		40120: 	
			SCREWING_RESULT:=E_TEST_STATE.PASSED;
			IF SCREWING_RESULT=E_TEST_STATE.PASSED THEN
				STATE:=40130;
			ELSE
				STATE:=40140;
			END_IF	
		40130:		(* Log NonConformance data *)
			IF MES.ASSY_SAVE_NCDAT(MRT_BARCODE, INDEX, NCDAT) THEN
				IF RESP.RESP_CODE = '0' THEN
					STATE:=40140;
				ELSE
					DEBUG:='40130 - SAVE_NCDAT() failed with wrong rescode';
					STATE:=99999;
				END_IF		
			END_IF
		40140:		(* Log Measurement data if failed *)
			IF MES.ASSY_SAVE_MESDAT(MRT_BARCODE, INDEX, MESDAT) THEN
				IF RESP.RESP_CODE = '0' THEN
					STATE:=40150;
				ELSE
					DEBUG:='40140 - SAVE_MESDAT() failed with wrong rescode';
					STATE:=99999;
				END_IF			
			END_IF		
			
		40150:		(* Complete OP_SCREWING_AUTO_2 in my case is index[10]. *)
			IF MES.COMPLETE_SFC(MRT_BARCODE, INDEX, SCREWING_RESULT) THEN
				IF RESP.RESP_CODE='0' THEN
					STATE:=50000;
				ELSE
					DEBUG:='40150 - ASSY_COMPLETE_SFC() failed with wrong rescode';
					STATE:=99999;
				END_IF
			END_IF
	
	80000:
			IF MES.START_SFC('288000000002010103983201', 1) THEN
				IF RESP.RESP_CODE='0' THEN
					STATE:=80100;
				ELSE
					DEBUG:='80000 - ASSY_START_SFC() failed with wrong rescode';
					STATE:=99999;
				END_IF
			END_IF
	80100: 		(* Get ricpe name *)
		IF MES.GET_RECIPE_NAME_BY_OPERATION_JSON('OP_GAP_FILLER_CHECK_COVER', GAP_FILLER_CHECK_RECIPE) THEN
			IF GAP_FILLER_CHECK_RECIPE<>'' THEN
				STATE:=80300;
			ELSE
				DEBUG:='20010 - GET_RECIPE_NAME_BY_OPERATION_JSON() failed with wrong rescode or empty recipe';
				STATE:=80200;
			END_IF
		END_IF
	
	END_CASE	
END_IF

FB_CALL_ACT();

ACTION FB_CALL_ACT:
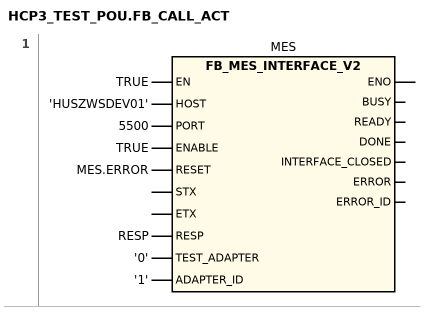
// NETWORK 1
MES(
    HOST := 'HUSZWSDEV01',
    PORT := 5500,
    ENABLE := TRUE,
    RESET := MES.ERROR,
    RESP := RESP,
    TEST_ADAPTER := '0',
    ADAPTER_ID := '1'); // FB_MES_INTERFACE_V2
END_ACTION

END_PROGRAM

// TESTs/TEST_POU_1026_REPAIR
PROGRAM TEST_POU_1026_REPAIR
VAR
	MES:						FB_MES_INTERFACE_V2;		(* Instance of MES-Interface function block *)
	RESP:						ST_REQUEST;				(* Reference to MES-Interface function block response *)
	INIT:						BOOL:=TRUE;
	RESET:						BOOL;					
	START:						BOOL;					
	STATE:						UDINT;
	INDEX:						INT;					
	
	BARCODE:					STRING:='288000060010020103725571';					(* COVER barcode *)
	OP_STATE:					ST_GET_OP_STATE;		(* Container of SFC State data which releated to Cover barcode *)					
	
	DEBUG:						STRING(255);
	EXIT_INTERFACE:				BOOL;
	SHOW_INTERFACE:				BOOL;
	HIDE_INTERFACE:				BOOL;
END_VAR

IF INIT THEN
	(* Restart the SAP-ME Interface.exe on PLC restart. Or triggered on strange communication error. 
	IF MES.LOCAL_INIT_SERVICE() THEN
		INIT:=FALSE;
	END_IF
	*)
	IF MES.GET_SERVICE_CONFIG() THEN
		INIT:=FALSE;
	END_IF
ELSE
	IF EXIT_INTERFACE THEN
		(* TCP Request for exiting. *)
		IF MES.EXIT_SERVICE() THEN
			EXIT_INTERFACE:=FALSE;
		END_IF
	END_IF
	IF SHOW_INTERFACE THEN
		IF MES.SHOW_SERVICE() THEN
			SHOW_INTERFACE:=FALSE;
		END_IF
	END_IF
	IF HIDE_INTERFACE THEN
		IF MES.HIDE_SERVICE() THEN
			HIDE_INTERFACE:=FALSE;
		END_IF
	END_IF
	CASE STATE OF
	(* ###############################################################		Initialize		###########################################################################	*)

	(* ###############################################################		Wait for start	###########################################################################	*)
		0:		(* Wait the start trigger *)
			IF START THEN
				INDEX:=0;
				STATE:=1000;
				START:=FALSE;
			END_IF				
	(* ################################################################################################################################################################
	   #
	   #
	   #																	ST10-Manual insertion
	   #
	   #
	   ################################################################################################################################################################ *)
	(* ###############################################################		Cover	insert	###########################################################################	*)
		1000:		(* Get current operation state of the cover *)
			IF MES.GET_CURRENT_OPERATION_STATE(BARCODE, INDEX, OP_STATE) THEN 
				IF RESP.RESP_CODE='0' OR RESP.RESP_CODE='377' THEN
					STATE:=99999;
				ELSE
					DEBUG:='1000 - GET_OP_STATE() failed with wrong rescode';
					STATE:=99999;
				END_IF
			END_IF

	END_CASE	
END_IF

FB_CALL_ACT();

ACTION FB_CALL_ACT:
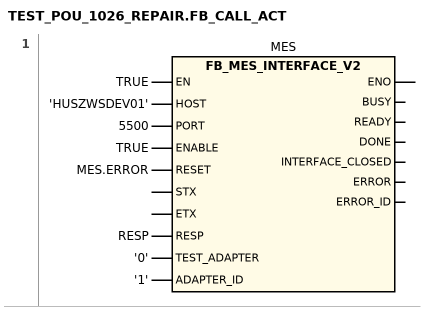
// NETWORK 1
MES(
    HOST := 'HUSZWSDEV01',
    PORT := 5500,
    ENABLE := TRUE,
    RESET := MES.ERROR,
    RESP := RESP,
    TEST_ADAPTER := '0',
    ADAPTER_ID := '1'); // FB_MES_INTERFACE_V2
END_ACTION

END_PROGRAM

// TESTs/TEST_POU_3026_SAVE_CF
PROGRAM TEST_POU_3026_SAVE_CF
VAR
	MES:						FB_MES_INTERFACE_V2;		(* Instance of MES-Interface function block *)
	RESP:						ST_REQUEST;				(* Reference to MES-Interface function block response *)
	INIT:						BOOL:=TRUE;
	RESET:						BOOL;					
	START:						BOOL;					
	STATE:						UDINT;
	INDEX:						INT:=0;					
	TEST_STATE:					INT:=0;
	BARCODE:					STRING:='380039001016010202222222';					(* valid barcode *)
	ADAPTERID:					STRING:='0';
	CF_NAME:					STRING:='ECUUID'; (* Custom field NAME TODO? KEY*)
	CF_VALUE:					STRING:='Test from PLC'; (* Custom field TODO: VALUE: VALUE *)	
	DEBUG:						STRING(255):='';
	EXIT_INTERFACE:				BOOL;
	SHOW_INTERFACE:				BOOL;
	HIDE_INTERFACE:				BOOL;
END_VAR

IF INIT THEN
	(* Restart the SAP-ME Interface.exe on PLC restart. Or triggered on strange communication error. 
	IF MES.LOCAL_INIT_SERVICE() THEN
		INIT:=FALSE;
	END_IF
	*)
	IF MES.GET_SERVICE_CONFIG() THEN
		INIT:=FALSE;
	END_IF
ELSE

	CASE STATE OF
	(* ###############################################################		Initialize		###########################################################################	*)

	(* ###############################################################		Wait for start	###########################################################################	*)
		0:		(* Wait the start trigger *)
			IF START THEN
				INDEX:=0;
				STATE:=2000;
				START:=FALSE;
				DEBUG:='';
			END_IF				

		2000:		(* START *) (* START and COMPLETE is necessary!!*)

			IF MES.START_SFC(BARCODE, INDEX) THEN
				IF RESP.RESP_CODE='0' THEN
					STATE:= 2001;
					DEBUG:= CONCAT(DEBUG,'2000 - START_SFC() OK ');					
				ELSE
					DEBUG:= CONCAT(DEBUG, '2000 - START_SFC() failed with wrong rescode ');
				END_IF
			ELSE
				DEBUG:= CONCAT(DEBUG, '2000 - START_SFC() started but not done yet ');
			END_IF
		2001: (* SAVE Custom field*)
				IF MES.SAVE_SFC_DATA(BARCODE,ADAPTERID, INDEX, CF_NAME,CF_VALUE) THEN 
					IF RESP.RESP_CODE='0' THEN
						DEBUG:= CONCAT(DEBUG,'2001 - SAVE_SFC_DATA() OK ');
						STATE:= 2002;					
					ELSE
						DEBUG:=CONCAT(DEBUG,'2001 - SAVE_SFC_DATA() failed ');
						STATE:=99999;
					END_IF
				ELSE
					DEBUG:= CONCAT(DEBUG,'2001 - SAVE_SFC_DATA() started but is not done ');
				END_IF
		2002: (* Complete *)
			IF MES.COMPLETE_SFC(BARCODE, INDEX, TEST_STATE) THEN
					IF RESP.RESP_CODE='0' THEN
						DEBUG:= CONCAT(DEBUG,'2002 - COMPLETE_SFC() OK ');
						STATE:=99999;					
					ELSE
						DEBUG:=CONCAT(DEBUG,'2002 - COMPLETE_SFC() failed with wrong rescode ');
						STATE:=99999;
					END_IF
			ELSE
				DEBUG:=CONCAT(DEBUG,'2002 - COMPLETE_SFC() started but not done yet. ');
			END_IF
	END_CASE	
END_IF
FB_CALL_ACT();

ACTION FB_CALL_ACT:
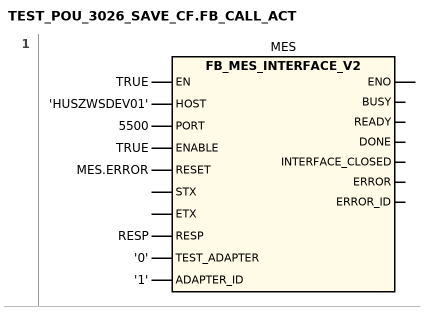
// NETWORK 1
MES(
    HOST := 'HUSZWSDEV01',
    PORT := 5500,
    ENABLE := TRUE,
    RESET := MES.ERROR,
    RESP := RESP,
    TEST_ADAPTER := '0',
    ADAPTER_ID := '1'); // FB_MES_INTERFACE_V2
END_ACTION

END_PROGRAM
